// §3.8a probe recipe record: the probe root's own model data.
TYPE ST_ProbeModelParCfg :
STRUCT
    SchemaVersion : UINT := 1;
    Speed         : DINT;
END_STRUCT
END_TYPE

(* stored: Version 1.1.0.1, ProductVersion 3.1.4024.12
   DUT ST_ProbeModelParCfg: Id {8d4f2a61-3b9e-4c07-a5d2-7e1c9b0f6a38} *)
